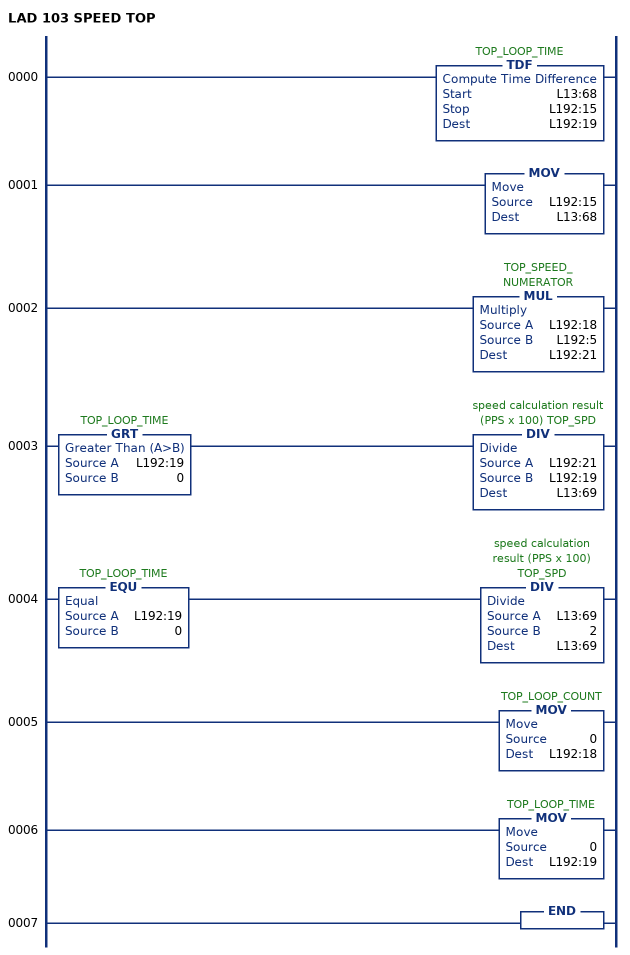
% Rung: 0 %
SOR TDF L13:68 L192:15 L192:19 EOR
%   L192:15  TOP_THIS_TIME  "rtc top belt movement event time" %
%   L192:19  TOP_LOOP_TIME %
% Rung: 1 %
SOR MOV L192:15 L13:68 EOR
%   L192:15  TOP_THIS_TIME  "rtc top belt movement event time" %
% Rung: 2 %
SOR MUL L192:18 L192:5 L192:21 EOR
%   L192:18  TOP_LOOP_COUNT %
%   L192:5  TKS_PER_SECOND %
%   L192:21  TOP_SPEED_NUMERATOR %
% Rung: 3 %
SOR GRT L192:19 0 DIV L192:21 L192:19 L13:69 EOR
%   L192:19  TOP_LOOP_TIME %
%   L192:21  TOP_SPEED_NUMERATOR %
%   L13:69  TOP_SPD  "speed calculation result (PPS x 100)" %
% Rung: 4 %
SOR EQU L192:19 0 DIV L13:69 2 L13:69 EOR
%   L192:19  TOP_LOOP_TIME %
%   L13:69  TOP_SPD  "speed calculation result (PPS x 100)" %
% Rung: 5 %
SOR MOV 0 L192:18 EOR
%   L192:18  TOP_LOOP_COUNT %
% Rung: 6 %
SOR MOV 0 L192:19 EOR
%   L192:19  TOP_LOOP_TIME %
% Rung: 7 %
SOR END EOR

LADDER 105 "P TOP"    % high speed %
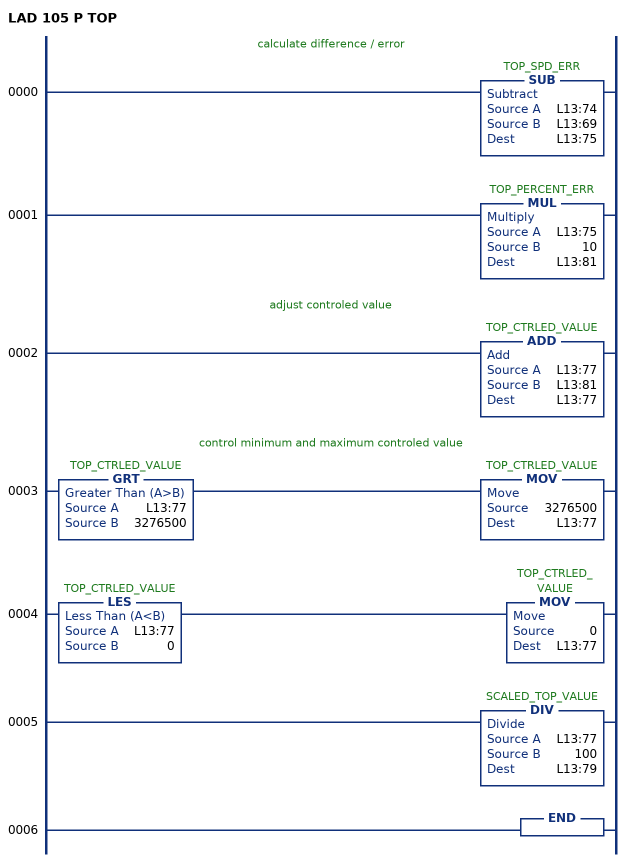
% Rung: 0 %
% calculate difference / error %
SOR SUB L13:74 L13:69 L13:75 EOR
%   L13:74  TOP_SPD_SETPOINT %
%   L13:69  TOP_SPD  "speed calculation result (PPS x 100)" %
%   L13:75  TOP_SPD_ERR %
% Rung: 1 %
SOR MUL L13:75 10 L13:81 EOR
%   L13:75  TOP_SPD_ERR %
%   L13:81  TOP_PERCENT_ERR %
% Rung: 2 %
% adjust controled value %
SOR ADD L13:77 L13:81 L13:77 EOR
%   L13:77  TOP_CTRLED_VALUE %
%   L13:81  TOP_PERCENT_ERR %
% Rung: 3 %
% control minimum and maximum controled value %
SOR GRT L13:77 3276500 MOV 3276500 L13:77 EOR
%   L13:77  TOP_CTRLED_VALUE %
% Rung: 4 %
SOR LES L13:77 0 MOV 0 L13:77 EOR
%   L13:77  TOP_CTRLED_VALUE %
% Rung: 5 %
SOR DIV L13:77 100 L13:79 EOR
%   L13:77  TOP_CTRLED_VALUE %
%   L13:79  SCALED_TOP_VALUE %
% Rung: 6 %
SOR END EOR

LADDER 111 "SHIFT TOP"
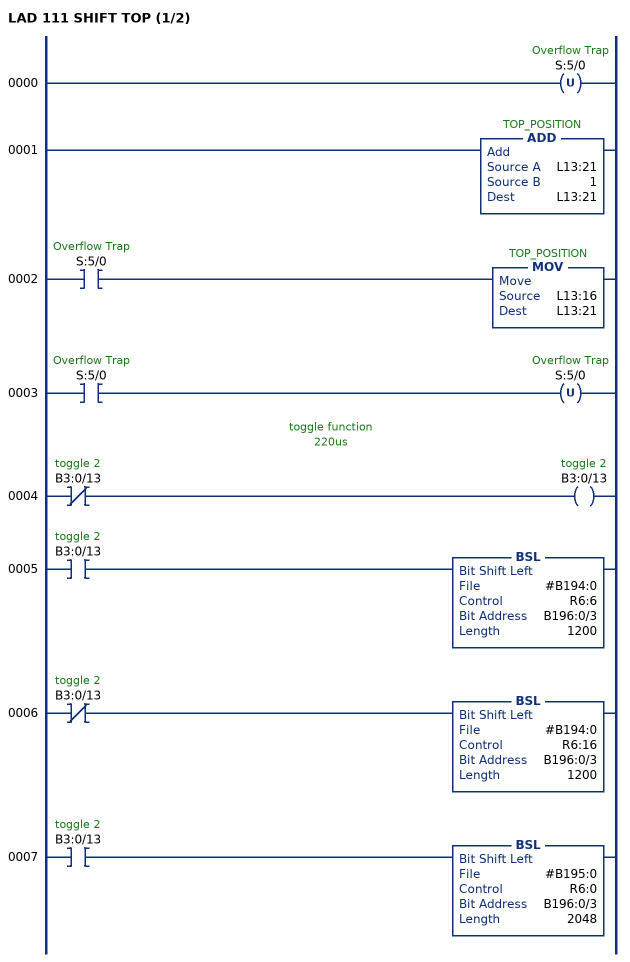
% Rung: 0 %
SOR OTU S:5/0 EOR
%   S:5/0  "Overflow Trap" %
% Rung: 1 %
SOR ADD L13:21 1 L13:21 EOR
%   L13:21  TOP_POSITION %
% Rung: 2 %
SOR XIC S:5/0 MOV L13:16 L13:21 EOR
%   S:5/0  "Overflow Trap" %
%   L13:16  MIN_LONG %
%   L13:21  TOP_POSITION %
% Rung: 3 %
SOR XIC S:5/0 OTU S:5/0 EOR
%   S:5/0  "Overflow Trap" %
% Rung: 4 %
% toggle function
% 220us %
SOR XIO B3:0/13 OTE B3:0/13 EOR
%   B3:0/13  "toggle 2" %
% Rung: 5 %
SOR XIC B3:0/13 BSL #B194:0 R6:6 B196:0/3 1200 EOR
%   B3:0/13  "toggle 2" %
%   R6:6  "from top load to top optic" %
%   B196:0/3  OFF %
% Rung: 6 %
SOR XIO B3:0/13 BSL #B194:0 R6:16 B196:0/3 1200 EOR
%   B3:0/13  "toggle 2" %
%   B196:0/3  OFF %
% Rung: 7 %
SOR XIC B3:0/13 BSL #B195:0 R6:0 B196:0/3 2048 EOR
%   B3:0/13  "toggle 2" %
%   B196:0/3  OFF %

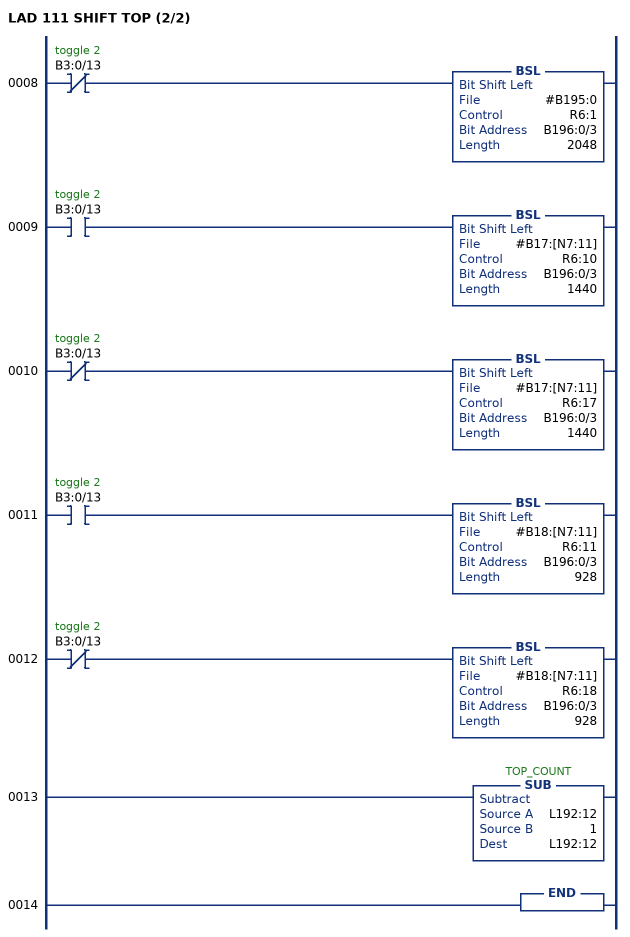
% Rung: 8 %
SOR XIO B3:0/13 BSL #B195:0 R6:1 B196:0/3 2048 EOR
%   B3:0/13  "toggle 2" %
%   B196:0/3  OFF %
% Rung: 9 %
SOR XIC B3:0/13 BSL #B17:[N7:11] R6:10 B196:0/3 1440 EOR
%   B3:0/13  "toggle 2" %
%   B196:0/3  OFF %
% Rung: 10 %
SOR XIO B3:0/13 BSL #B17:[N7:11] R6:17 B196:0/3 1440 EOR
%   B3:0/13  "toggle 2" %
%   B196:0/3  OFF %
% Rung: 11 %
SOR XIC B3:0/13 BSL #B18:[N7:11] R6:11 B196:0/3 928 EOR
%   B3:0/13  "toggle 2" %
%   B196:0/3  OFF %
% Rung: 12 %
SOR XIO B3:0/13 BSL #B18:[N7:11] R6:18 B196:0/3 928 EOR
%   B3:0/13  "toggle 2" %
%   B196:0/3  OFF %
% Rung: 13 %
SOR SUB L192:12 1 L192:12 EOR
%   L192:12  TOP_COUNT %
% Rung: 14 %
SOR END EOR

LADDER 131 "READXFER"
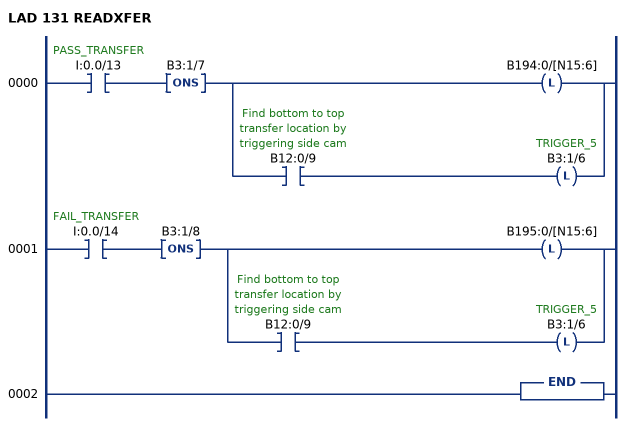
% Rung: 0 %
SOR XIC I:0.0/13 ONS B3:1/7 BST OTL B194:0/[N15:6] NXB XIC B12:0/9 OTL B3:1/6 BND EOR
%   I:0.0/13  PASS_TRANSFER %
%   N15:6  XFER_IN_LOC %
%   B12:0/9  "Find bottom to top transfer location by triggering side cam" %
%   B3:1/6  TRIGGER_5 %
% Rung: 1 %
SOR XIC I:0.0/14 ONS B3:1/8 BST OTL B195:0/[N15:6] NXB XIC B12:0/9 OTL B3:1/6 BND EOR
%   I:0.0/14  FAIL_TRANSFER %
%   N15:6  XFER_IN_LOC %
%   B12:0/9  "Find bottom to top transfer location by triggering side cam" %
%   B3:1/6  TRIGGER_5 %
% Rung: 2 %
SOR END EOR

LADDER 140 "TOP_OPTIC"
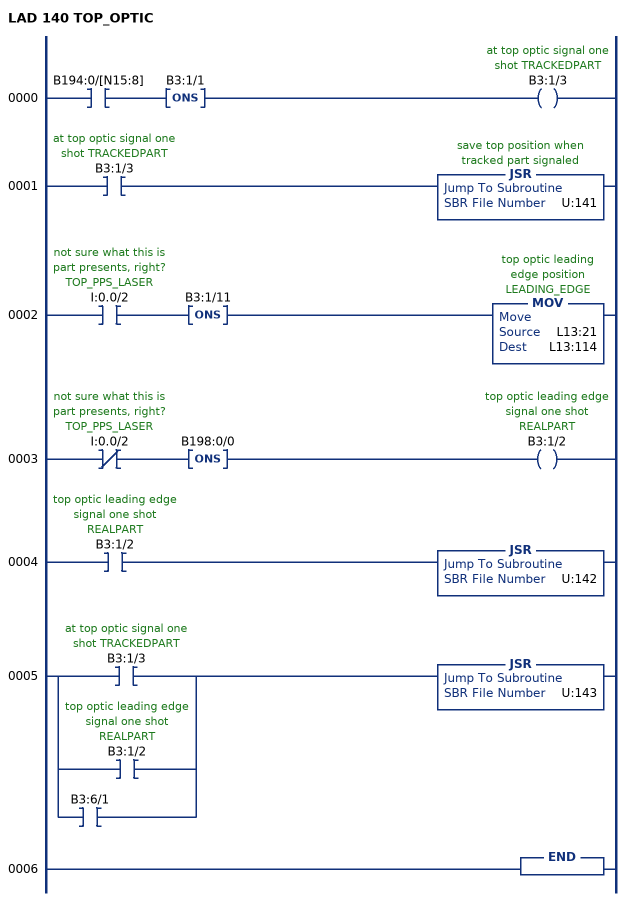
% Rung: 0 %
SOR XIC B194:0/[N15:8] ONS B3:1/1 OTE B3:1/3 EOR
%   N15:8  TOP_OPTIC_LOC %
%   B3:1/3  TRACKEDPART  "at top optic signal one shot" %
% Rung: 1 %
SOR XIC B3:1/3 JSR U:141 EOR
%   B3:1/3  TRACKEDPART  "at top optic signal one shot" %
%   U:141  "save top position when tracked part signaled" %
% Rung: 2 %
SOR XIC I:0.0/2 ONS B3:1/11 MOV L13:21 L13:114 EOR
%   I:0.0/2  TOP_PPS_LASER  "not sure what this is part presents, right?" %
%   L13:21  TOP_POSITION %
%   L13:114  LEADING_EDGE  "top optic leading edge position" %
% Rung: 3 %
SOR XIO I:0.0/2 ONS B198:0/0 OTE B3:1/2 EOR
%   I:0.0/2  TOP_PPS_LASER  "not sure what this is part presents, right?" %
%   B3:1/2  REALPART  "top optic leading edge signal one shot" %
% Rung: 4 %
SOR XIC B3:1/2 JSR U:142 EOR
%   B3:1/2  REALPART  "top optic leading edge signal one shot" %
% Rung: 5 %
SOR BST XIC B3:1/3 NXB XIC B3:1/2 NXB XIC B3:6/1 BND JSR U:143 EOR
%   B3:1/3  TRACKEDPART  "at top optic signal one shot" %
%   B3:1/2  REALPART  "top optic leading edge signal one shot" %
% Rung: 6 %
SOR END EOR

LADDER 141 "TOPOP_VERT"
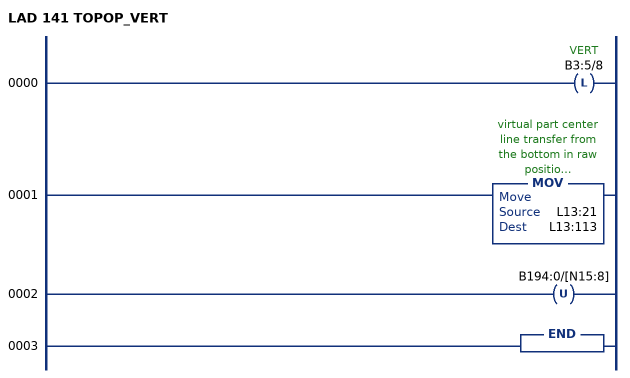
% Rung: 0 %
SOR OTL B3:5/8 EOR
%   B3:5/8  VERT %
% Rung: 1 %
SOR MOV L13:21 L13:113 EOR
%   L13:21  TOP_POSITION %
%   L13:113  VERTUAL_PT_RAW_CL  "virtual part center line transfer from the bottom in raw position" %
% Rung: 2 %
SOR OTU B194:0/[N15:8] EOR
%   N15:8  TOP_OPTIC_LOC %
% Rung: 3 %
SOR END EOR

LADDER 142 "TOPOP_REAL"
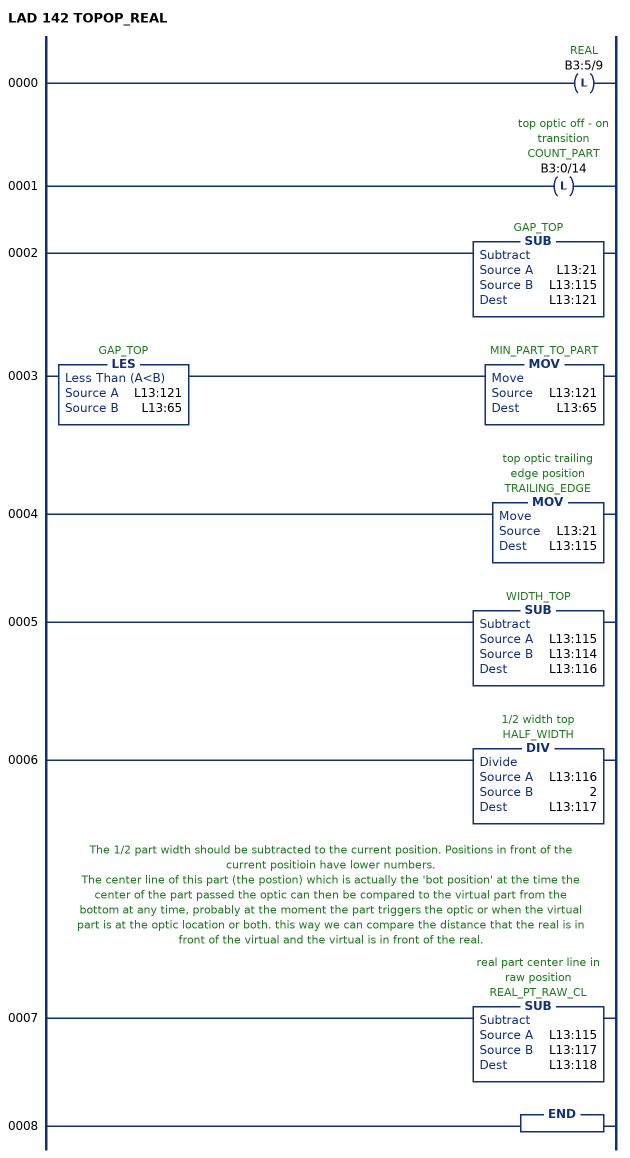
% Rung: 0 %
SOR OTL B3:5/9 EOR
%   B3:5/9  REAL %
% Rung: 1 %
SOR OTL B3:0/14 EOR
%   B3:0/14  COUNT_PART  "top optic off - on transition" %
% Rung: 2 %
SOR SUB L13:21 L13:115 L13:121 EOR
%   L13:21  TOP_POSITION %
%   L13:115  TRAILING_EDGE  "top optic trailing edge position" %
%   L13:121  GAP_TOP %
% Rung: 3 %
SOR LES L13:121 L13:65 MOV L13:121 L13:65 EOR
%   L13:121  GAP_TOP %
%   L13:65  MIN_PART_TO_PART %
% Rung: 4 %
SOR MOV L13:21 L13:115 EOR
%   L13:21  TOP_POSITION %
%   L13:115  TRAILING_EDGE  "top optic trailing edge position" %
% Rung: 5 %
SOR SUB L13:115 L13:114 L13:116 EOR
%   L13:115  TRAILING_EDGE  "top optic trailing edge position" %
%   L13:114  LEADING_EDGE  "top optic leading edge position" %
%   L13:116  WIDTH_TOP %
% Rung: 6 %
SOR DIV L13:116 2 L13:117 EOR
%   L13:116  WIDTH_TOP %
%   L13:117  HALF_WIDTH  "1/2 width top" %
% Rung: 7 %
% The 1/2 part width should be subtracted to the current position. Positions in front of the current positioin have lower numbers.
% 
% The center line of this part (the postion) which is actually the 'bot position' at the time the center of the part passed the optic can then be compared to the virtual part from the bottom at any time, probably at the moment the part triggers the optic or when the virtual part is at the optic location or both. this way we can compare the distance that the real is in front of the virtual and the virtual is in front of the real. %
SOR SUB L13:115 L13:117 L13:118 EOR
%   L13:115  TRAILING_EDGE  "top optic trailing edge position" %
%   L13:117  HALF_WIDTH  "1/2 width top" %
%   L13:118  REAL_PT_RAW_CL  "real part center line in raw position" %
% Rung: 8 %
SOR END EOR

LADDER 143 "TOPOP_TEST"
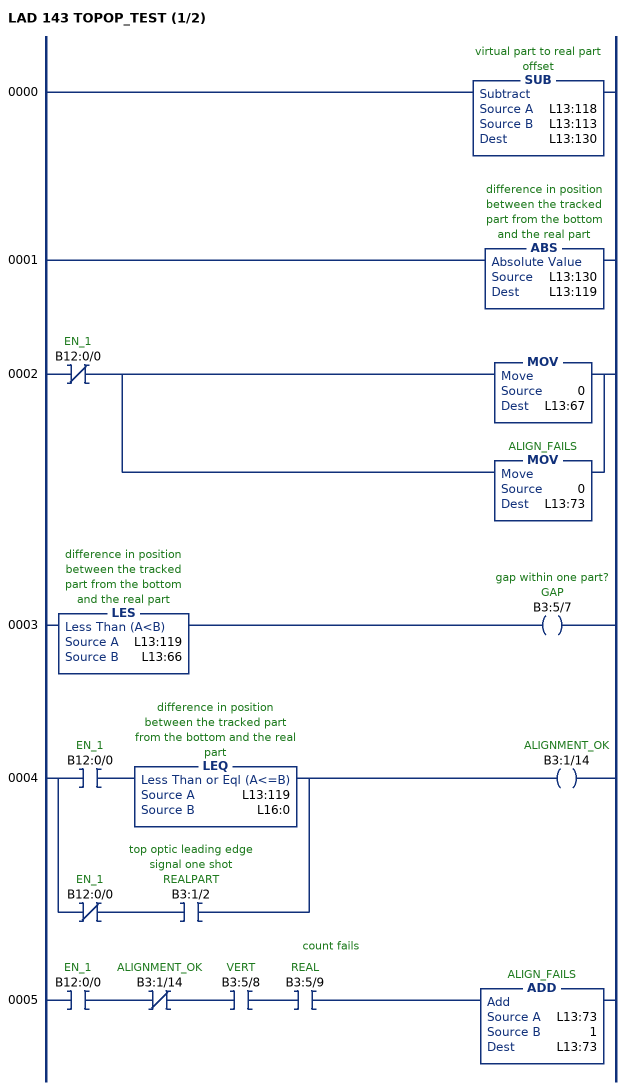
% Rung: 0 %
SOR SUB L13:118 L13:113 L13:130 EOR
%   L13:118  REAL_PT_RAW_CL  "real part center line in raw position" %
%   L13:113  VERTUAL_PT_RAW_CL  "virtual part center line transfer from the bottom in raw position" %
%   L13:130  "virtual part to real part offset" %
% Rung: 1 %
SOR ABS L13:130 L13:119 EOR
%   L13:130  "virtual part to real part offset" %
%   L13:119  "difference in position between the tracked part from the bottom and the real part" %
% Rung: 2 %
SOR XIO B12:0/0 BST MOV 0 L13:67 NXB MOV 0 L13:73 BND EOR
%   B12:0/0  EN_1 %
%   L13:73  ALIGN_FAILS %
% Rung: 3 %
SOR LES L13:119 L13:66 OTE B3:5/7 EOR
%   L13:119  "difference in position between the tracked part from the bottom and the real part" %
%   L13:66  SAME_PART_GAP %
%   B3:5/7  GAP  "gap within one part?" %
% Rung: 4 %
SOR BST XIC B12:0/0 LEQ L13:119 L16:0 NXB XIO B12:0/0 XIC B3:1/2 BND OTE B3:1/14 EOR
%   B12:0/0  EN_1 %
%   L13:119  "difference in position between the tracked part from the bottom and the real part" %
%   L16:0  MAX_OFFSET %
%   B3:1/2  REALPART  "top optic leading edge signal one shot" %
%   B3:1/14  ALIGNMENT_OK %
% Rung: 5 %
% count fails %
SOR XIC B12:0/0 XIO B3:1/14 XIC B3:5/8 XIC B3:5/9 ADD L13:73 1 L13:73 EOR
%   B12:0/0  EN_1 %
%   B3:1/14  ALIGNMENT_OK %
%   B3:5/8  VERT %
%   B3:5/9  REAL %
%   L13:73  ALIGN_FAILS %

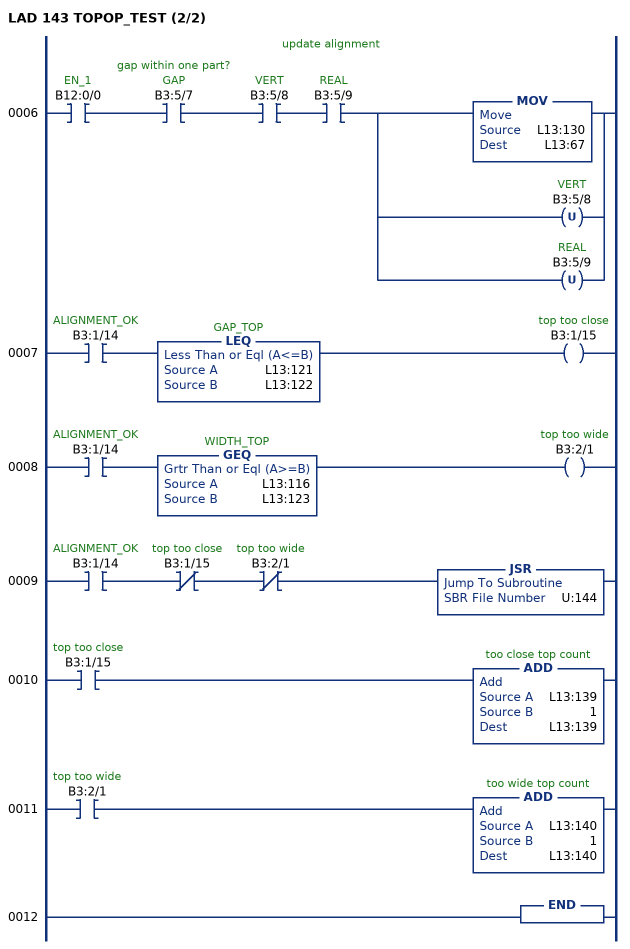
% Rung: 6 %
% update alignment %
SOR XIC B12:0/0 XIC B3:5/7 XIC B3:5/8 XIC B3:5/9 BST MOV L13:130 L13:67 NXB OTU B3:5/8 NXB OTU B3:5/9 BND EOR
%   B12:0/0  EN_1 %
%   B3:5/7  GAP  "gap within one part?" %
%   B3:5/8  VERT %
%   B3:5/9  REAL %
%   L13:130  "virtual part to real part offset" %
% Rung: 7 %
SOR XIC B3:1/14 LEQ L13:121 L13:122 OTE B3:1/15 EOR
%   B3:1/14  ALIGNMENT_OK %
%   L13:121  GAP_TOP %
%   L13:122  MIN_GAP_TOP %
%   B3:1/15  "top too close" %
% Rung: 8 %
SOR XIC B3:1/14 GEQ L13:116 L13:123 OTE B3:2/1 EOR
%   B3:1/14  ALIGNMENT_OK %
%   L13:116  WIDTH_TOP %
%   L13:123  MAX_WIDTH_TOP %
%   B3:2/1  "top too wide" %
% Rung: 9 %
SOR XIC B3:1/14 XIO B3:1/15 XIO B3:2/1 JSR U:144 EOR
%   B3:1/14  ALIGNMENT_OK %
%   B3:1/15  "top too close" %
%   B3:2/1  "top too wide" %
% Rung: 10 %
SOR XIC B3:1/15 ADD L13:139 1 L13:139 EOR
%   B3:1/15  "top too close" %
%   L13:139  "too close top count" %
% Rung: 11 %
SOR XIC B3:2/1 ADD L13:140 1 L13:140 EOR
%   B3:2/1  "top too wide" %
%   L13:140  "too wide top count" %
% Rung: 12 %
SOR END EOR

LADDER 144 "TOP_OP_OK"
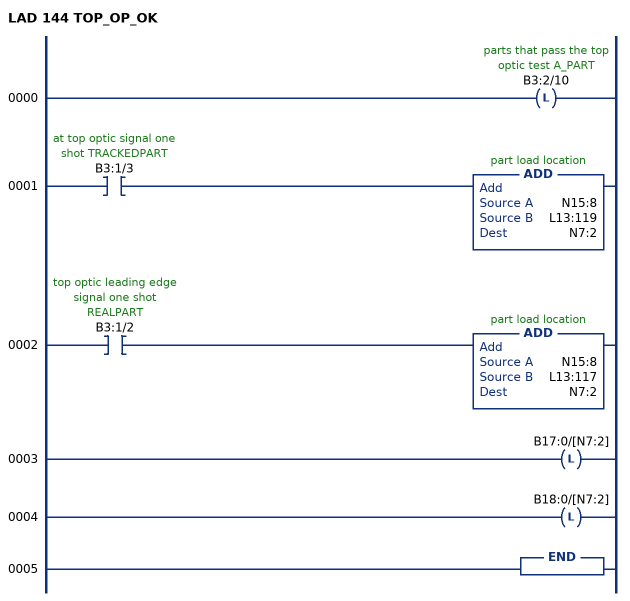
% Rung: 0 %
SOR OTL B3:2/10 EOR
%   B3:2/10  A_PART  "parts that pass the top optic test" %
% Rung: 1 %
SOR XIC B3:1/3 ADD N15:8 L13:119 N7:2 EOR
%   B3:1/3  TRACKEDPART  "at top optic signal one shot" %
%   N15:8  TOP_OPTIC_LOC %
%   L13:119  "difference in position between the tracked part from the bottom and the real part" %
%   N7:2  "part load location" %
% Rung: 2 %
SOR XIC B3:1/2 ADD N15:8 L13:117 N7:2 EOR
%   B3:1/2  REALPART  "top optic leading edge signal one shot" %
%   N15:8  TOP_OPTIC_LOC %
%   L13:117  HALF_WIDTH  "1/2 width top" %
%   N7:2  "part load location" %
% Rung: 3 %
SOR OTL B17:0/[N7:2] EOR
%   N7:2  "part load location" %
% Rung: 4 %
SOR OTL B18:0/[N7:2] EOR
%   N7:2  "part load location" %
% Rung: 5 %
SOR END EOR

LADDER 190 "INS5"
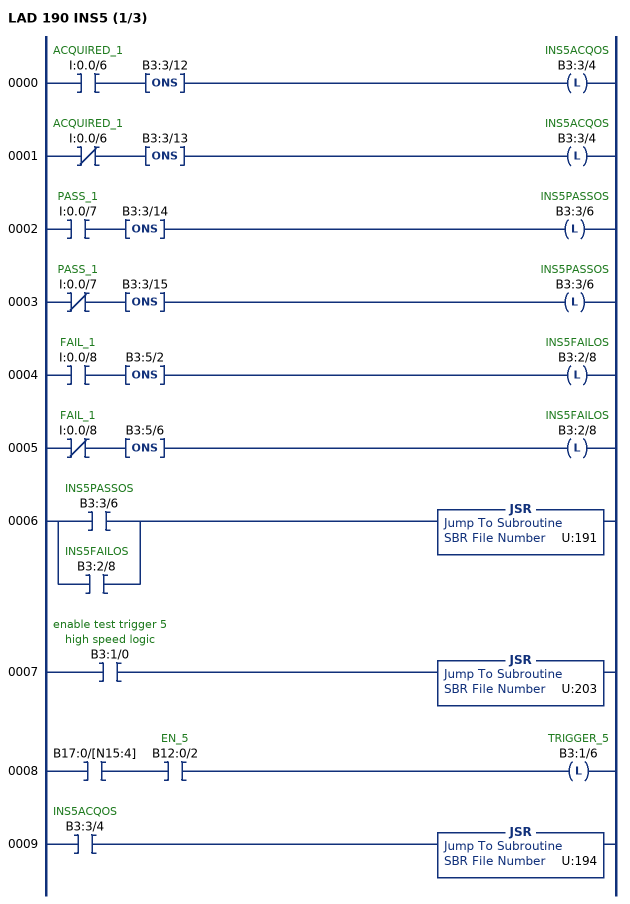
% Rung: 0 %
SOR XIC I:0.0/6 ONS B3:3/12 OTL B3:3/4 EOR
%   I:0.0/6  ACQUIRED_1 %
%   B3:3/4  INS5ACQOS %
% Rung: 1 %
SOR XIO I:0.0/6 ONS B3:3/13 OTL B3:3/4 EOR
%   I:0.0/6  ACQUIRED_1 %
%   B3:3/4  INS5ACQOS %
% Rung: 2 %
SOR XIC I:0.0/7 ONS B3:3/14 OTL B3:3/6 EOR
%   I:0.0/7  PASS_1 %
%   B3:3/6  INS5PASSOS %
% Rung: 3 %
SOR XIO I:0.0/7 ONS B3:3/15 OTL B3:3/6 EOR
%   I:0.0/7  PASS_1 %
%   B3:3/6  INS5PASSOS %
% Rung: 4 %
SOR XIC I:0.0/8 ONS B3:5/2 OTL B3:2/8 EOR
%   I:0.0/8  FAIL_1 %
%   B3:2/8  INS5FAILOS %
% Rung: 5 %
SOR XIO I:0.0/8 ONS B3:5/6 OTL B3:2/8 EOR
%   I:0.0/8  FAIL_1 %
%   B3:2/8  INS5FAILOS %
% Rung: 6 %
SOR BST XIC B3:3/6 NXB XIC B3:2/8 BND JSR U:191 EOR
%   B3:3/6  INS5PASSOS %
%   B3:2/8  INS5FAILOS %
% Rung: 7 %
SOR XIC B3:1/0 JSR U:203 EOR
%   B3:1/0  "enable test trigger 5 high speed logic" %
% Rung: 8 %
SOR XIC B17:0/[N15:4] XIC B12:0/2 OTL B3:1/6 EOR
%   N15:4  INS_5_TRIG_LOC %
%   B12:0/2  EN_5 %
%   B3:1/6  TRIGGER_5 %
% Rung: 9 %
SOR XIC B3:3/4 JSR U:194 EOR
%   B3:3/4  INS5ACQOS %

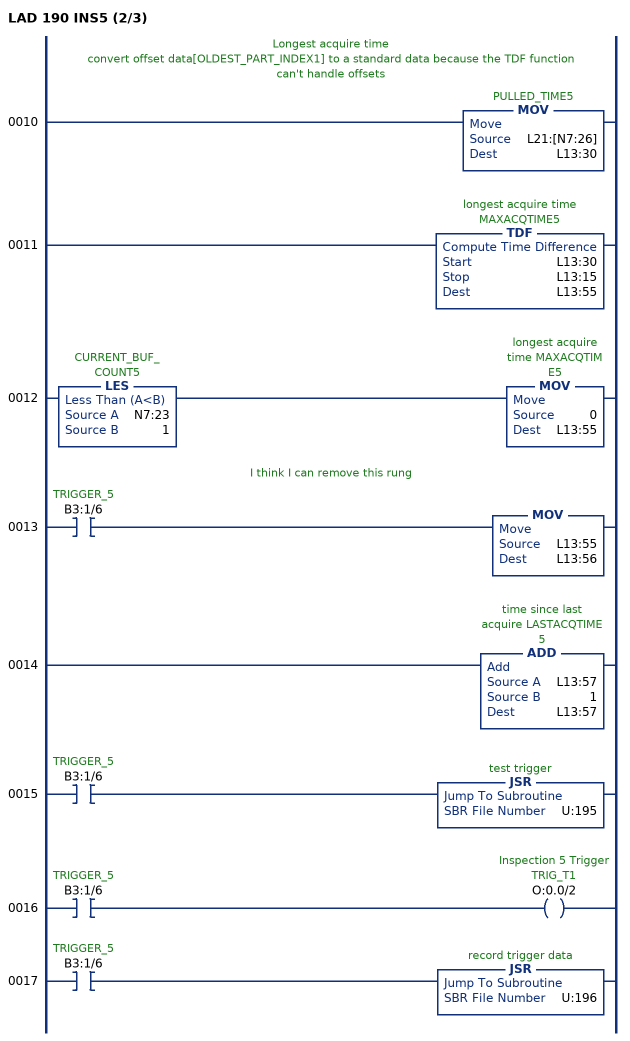
% Rung: 10 %
% Longest acquire time
% convert offset data[OLDEST_PART_INDEX1] to a standard data because the TDF function can't handle offsets %
SOR MOV L21:[N7:26] L13:30 EOR
%   N7:26  OLDEST_PART_INDEX5 %
%   L13:30  PULLED_TIME5 %
% Rung: 11 %
SOR TDF L13:30 L13:15 L13:55 EOR
%   L13:30  PULLED_TIME5 %
%   L13:15  TOP_TIME %
%   L13:55  MAXACQTIME5  "longest acquire time" %
% Rung: 12 %
SOR LES N7:23 1 MOV 0 L13:55 EOR
%   N7:23  CURRENT_BUF_COUNT5 %
%   L13:55  MAXACQTIME5  "longest acquire time" %
% Rung: 13 %
% I think I can remove this rung %
SOR XIC B3:1/6 MOV L13:55 L13:56 EOR
%   B3:1/6  TRIGGER_5 %
%   L13:55  MAXACQTIME5  "longest acquire time" %
% Rung: 14 %
SOR ADD L13:57 1 L13:57 EOR
%   L13:57  LASTACQTIME5  "time since last acquire" %
% Rung: 15 %
SOR XIC B3:1/6 JSR U:195 EOR
%   B3:1/6  TRIGGER_5 %
%   U:195  "test trigger" %
% Rung: 16 %
SOR XIC B3:1/6 OTE O:0.0/2 EOR
%   B3:1/6  TRIGGER_5 %
%   O:0.0/2  TRIG_T1  "Inspection 5 Trigger" %
% Rung: 17 %
SOR XIC B3:1/6 JSR U:196 EOR
%   B3:1/6  TRIGGER_5 %
%   U:196  "record trigger data" %

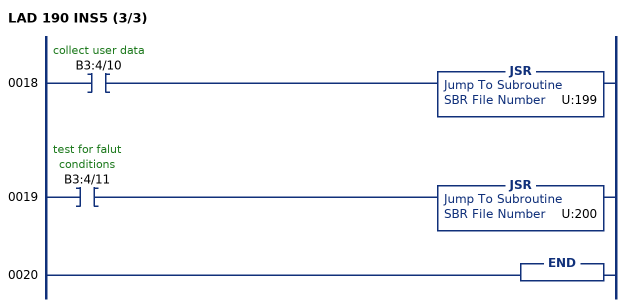
% Rung: 18 %
SOR XIC B3:4/10 JSR U:199 EOR
%   B3:4/10  "collect user data" %
% Rung: 19 %
SOR XIC B3:4/11 JSR U:200 EOR
%   B3:4/11  "test for falut conditions" %
% Rung: 20 %
SOR END EOR

LADDER 191 "INS5RESULT"
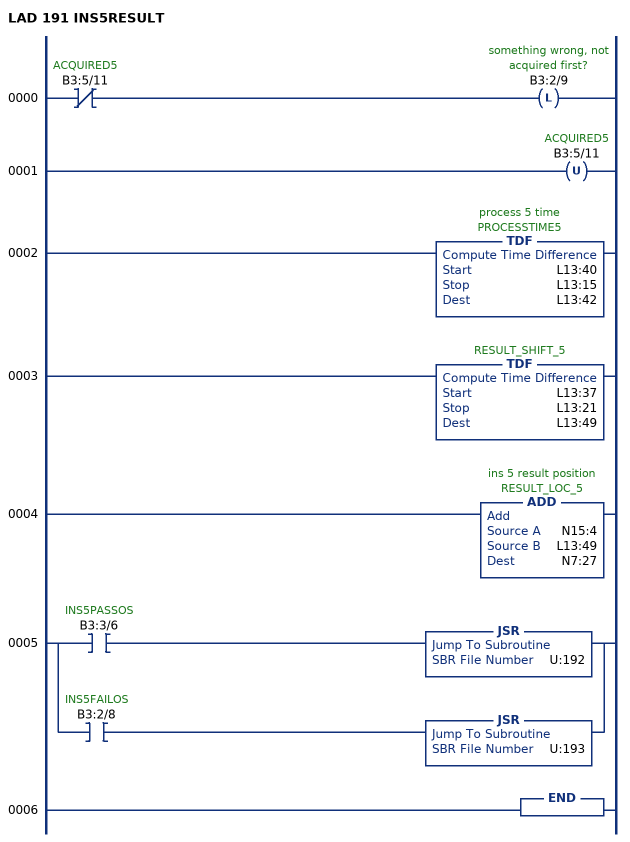
% Rung: 0 %
SOR XIO B3:5/11 OTL B3:2/9 EOR
%   B3:5/11  ACQUIRED5 %
%   B3:2/9  "something wrong, not acquired first?" %
% Rung: 1 %
SOR OTU B3:5/11 EOR
%   B3:5/11  ACQUIRED5 %
% Rung: 2 %
SOR TDF L13:40 L13:15 L13:42 EOR
%   L13:40  TIMEOFACQ5  "the time of the last acquire" %
%   L13:15  TOP_TIME %
%   L13:42  PROCESSTIME5  "process 5 time" %
% Rung: 3 %
SOR TDF L13:37 L13:21 L13:49 EOR
%   L13:37  PROCESS_START_POS_5 %
%   L13:21  TOP_POSITION %
%   L13:49  RESULT_SHIFT_5 %
% Rung: 4 %
SOR ADD N15:4 L13:49 N7:27 EOR
%   N15:4  INS_5_TRIG_LOC %
%   L13:49  RESULT_SHIFT_5 %
%   N7:27  RESULT_LOC_5  "ins 5 result position" %
% Rung: 5 %
SOR BST XIC B3:3/6 JSR U:192 NXB XIC B3:2/8 JSR U:193 BND EOR
%   B3:3/6  INS5PASSOS %
%   B3:2/8  INS5FAILOS %
% Rung: 6 %
SOR END EOR

LADDER 192 "INS5PASS"
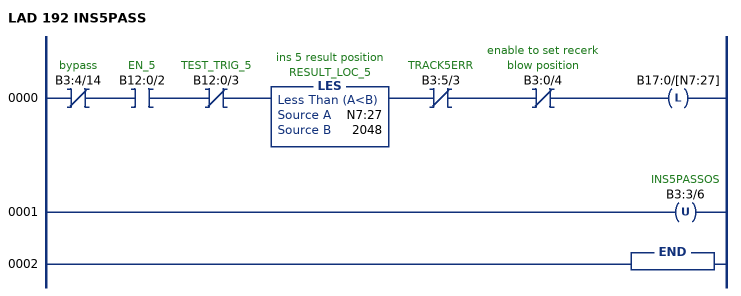
% Rung: 0 %
SOR XIO B3:4/14 XIC B12:0/2 XIO B12:0/3 LES N7:27 2048 XIO B3:5/3 XIO B3:0/4 OTL B17:0/[N7:27] EOR
%   B3:4/14  "bypass" %
%   B12:0/2  EN_5 %
%   B12:0/3  TEST_TRIG_5 %
%   N7:27  RESULT_LOC_5  "ins 5 result position" %
%   B3:5/3  TRACK5ERR %
%   B3:0/4  "enable to set recerk blow position" %
% Rung: 1 %
SOR OTU B3:3/6 EOR
%   B3:3/6  INS5PASSOS %
% Rung: 2 %
SOR END EOR

LADDER 193 "INS5FAIL"
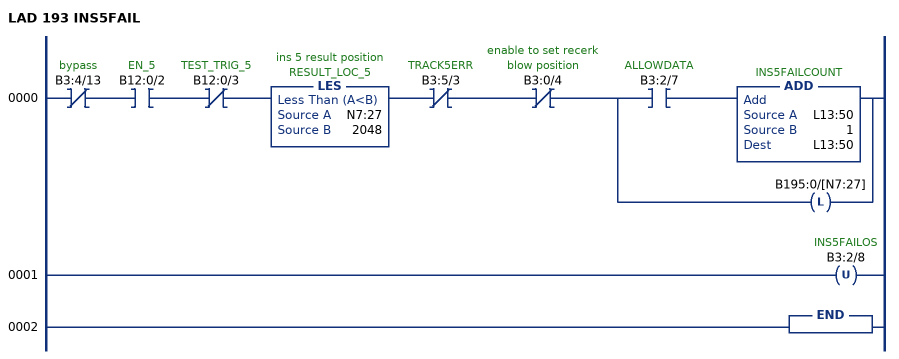
% Rung: 0 %
SOR XIO B3:4/13 XIC B12:0/2 XIO B12:0/3 LES N7:27 2048 XIO B3:5/3 XIO B3:0/4 BST XIC B3:2/7 ADD L13:50 1 L13:50 NXB OTL B195:0/[N7:27] BND EOR
%   B3:4/13  "bypass" %
%   B12:0/2  EN_5 %
%   B12:0/3  TEST_TRIG_5 %
%   N7:27  RESULT_LOC_5  "ins 5 result position" %
%   B3:5/3  TRACK5ERR %
%   B3:0/4  "enable to set recerk blow position" %
%   B3:2/7  ALLOWDATA %
%   L13:50  INS5FAILCOUNT %
% Rung: 1 %
SOR OTU B3:2/8 EOR
%   B3:2/8  INS5FAILOS %
% Rung: 2 %
SOR END EOR

LADDER 194 "INS5ACQ"
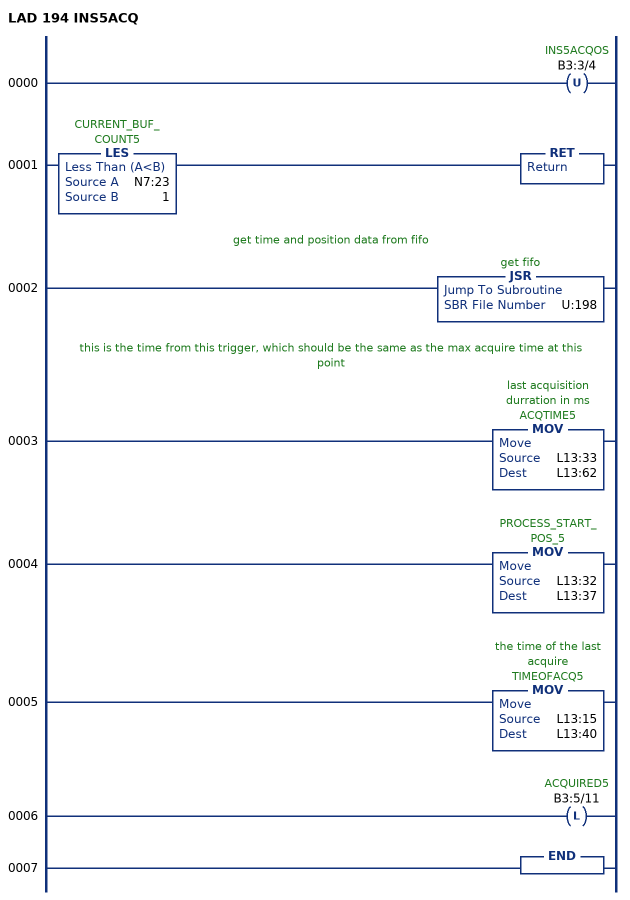
% Rung: 0 %
SOR OTU B3:3/4 EOR
%   B3:3/4  INS5ACQOS %
% Rung: 1 %
SOR LES N7:23 1 RET EOR
%   N7:23  CURRENT_BUF_COUNT5 %
% Rung: 2 %
% get time and position data from fifo %
SOR JSR U:198 EOR
%   U:198  "get fifo" %
% Rung: 3 %
% this is the time from this trigger, which should be the same as the max acquire time at this point %
SOR MOV L13:33 L13:62 EOR
%   L13:33  TIME_SPAN5 %
%   L13:62  ACQTIME5  "last acquisition durration in ms" %
% Rung: 4 %
SOR MOV L13:32 L13:37 EOR
%   L13:32  PULLED_POSITION5 %
%   L13:37  PROCESS_START_POS_5 %
% Rung: 5 %
SOR MOV L13:15 L13:40 EOR
%   L13:15  TOP_TIME %
%   L13:40  TIMEOFACQ5  "the time of the last acquire" %
% Rung: 6 %
SOR OTL B3:5/11 EOR
%   B3:5/11  ACQUIRED5 %
% Rung: 7 %
SOR END EOR

LADDER 195 "Q5TIMETEST"
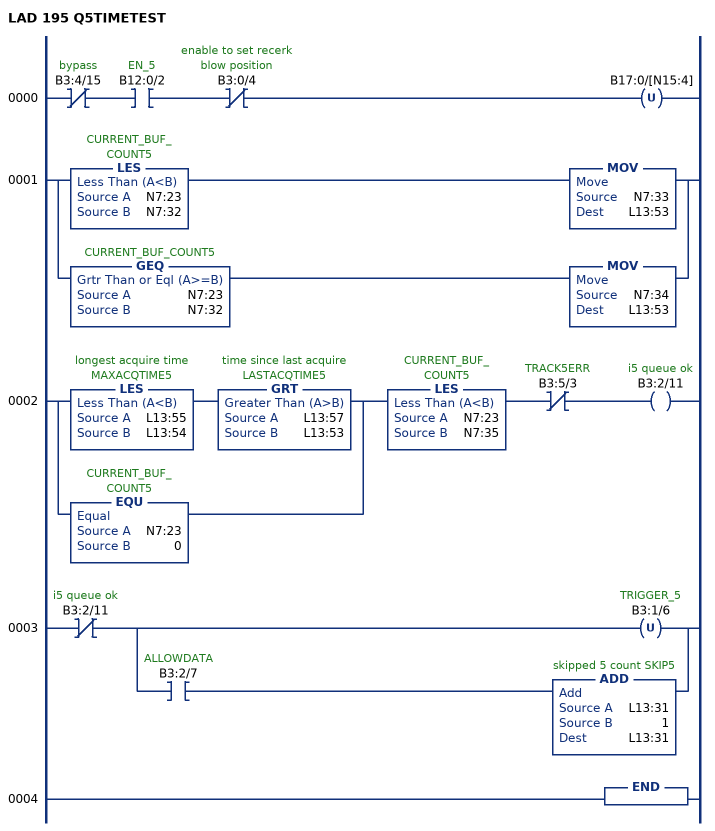
% Rung: 0 %
SOR XIO B3:4/15 XIC B12:0/2 XIO B3:0/4 OTU B17:0/[N15:4] EOR
%   B3:4/15  "bypass" %
%   B12:0/2  EN_5 %
%   B3:0/4  "enable to set recerk blow position" %
%   N15:4  INS_5_TRIG_LOC %
% Rung: 1 %
SOR BST LES N7:23 N7:32 MOV N7:33 L13:53 NXB GEQ N7:23 N7:32 MOV N7:34 L13:53 BND EOR
%   N7:23  CURRENT_BUF_COUNT5 %
% Rung: 2 %
SOR BST LES L13:55 L13:54 GRT L13:57 L13:53 NXB EQU N7:23 0 BND LES N7:23 N7:35 XIO B3:5/3 OTE B3:2/11 EOR
%   L13:55  MAXACQTIME5  "longest acquire time" %
%   L13:57  LASTACQTIME5  "time since last acquire" %
%   N7:23  CURRENT_BUF_COUNT5 %
%   N7:35  "maximum buffers" %
%   B3:5/3  TRACK5ERR %
%   B3:2/11  "i5 queue ok" %
% Rung: 3 %
SOR XIO B3:2/11 BST OTU B3:1/6 NXB XIC B3:2/7 ADD L13:31 1 L13:31 BND EOR
%   B3:2/11  "i5 queue ok" %
%   B3:1/6  TRIGGER_5 %
%   B3:2/7  ALLOWDATA %
%   L13:31  SKIP5  "skipped 5 count" %
% Rung: 4 %
SOR END EOR

LADDER 196 "INS5TRIG"
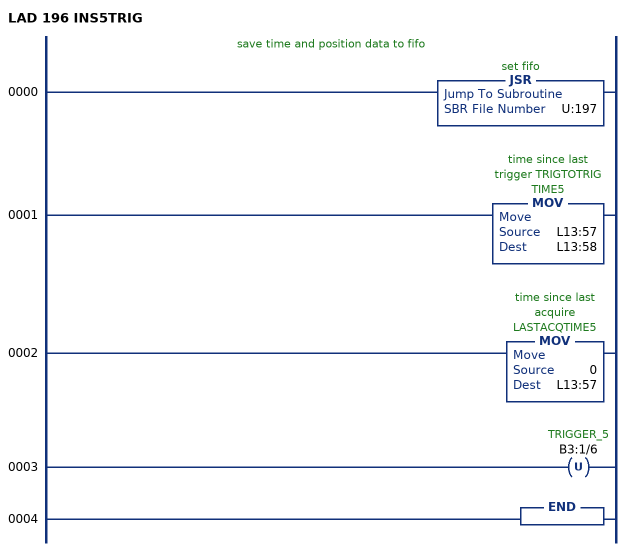
% Rung: 0 %
% save time and position data to fifo %
SOR JSR U:197 EOR
%   U:197  "set fifo" %
% Rung: 1 %
SOR MOV L13:57 L13:58 EOR
%   L13:57  LASTACQTIME5  "time since last acquire" %
%   L13:58  TRIGTOTRIGTIME5  "time since last trigger" %
% Rung: 2 %
SOR MOV 0 L13:57 EOR
%   L13:57  LASTACQTIME5  "time since last acquire" %
% Rung: 3 %
SOR OTU B3:1/6 EOR
%   B3:1/6  TRIGGER_5 %
% Rung: 4 %
SOR END EOR

LADDER 197 "FIFO5SET"
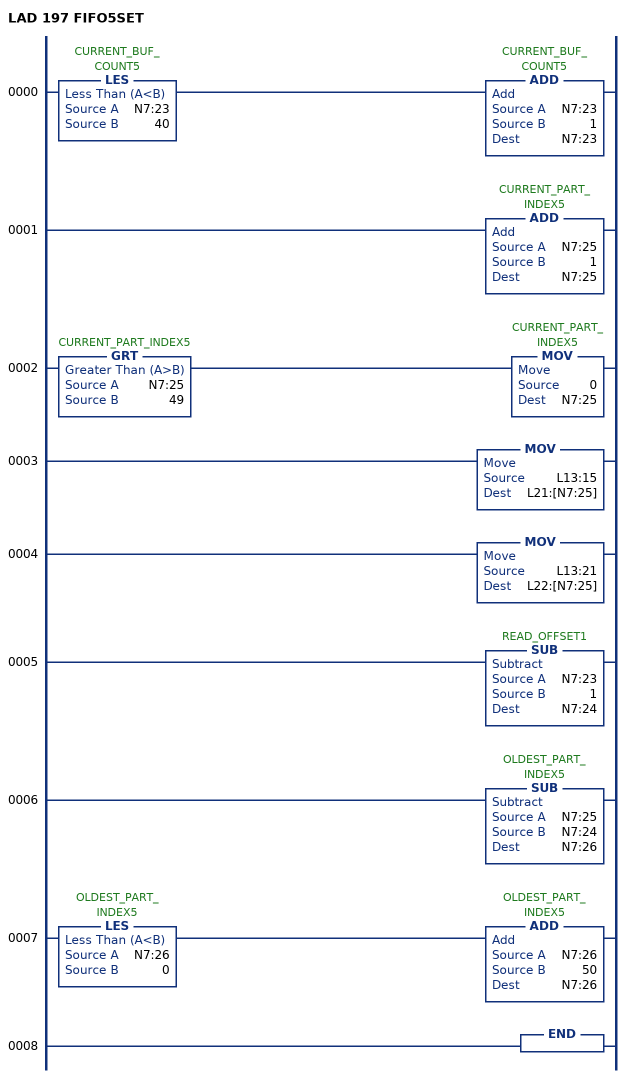
% Rung: 0 %
SOR LES N7:23 40 ADD N7:23 1 N7:23 EOR
%   N7:23  CURRENT_BUF_COUNT5 %
% Rung: 1 %
SOR ADD N7:25 1 N7:25 EOR
%   N7:25  CURRENT_PART_INDEX5 %
% Rung: 2 %
SOR GRT N7:25 49 MOV 0 N7:25 EOR
%   N7:25  CURRENT_PART_INDEX5 %
% Rung: 3 %
SOR MOV L13:15 L21:[N7:25] EOR
%   L13:15  TOP_TIME %
%   N7:25  CURRENT_PART_INDEX5 %
% Rung: 4 %
SOR MOV L13:21 L22:[N7:25] EOR
%   L13:21  TOP_POSITION %
%   N7:25  CURRENT_PART_INDEX5 %
% Rung: 5 %
SOR SUB N7:23 1 N7:24 EOR
%   N7:23  CURRENT_BUF_COUNT5 %
%   N7:24  "READ_OFFSET1" %
% Rung: 6 %
SOR SUB N7:25 N7:24 N7:26 EOR
%   N7:25  CURRENT_PART_INDEX5 %
%   N7:24  "READ_OFFSET1" %
%   N7:26  OLDEST_PART_INDEX5 %
% Rung: 7 %
SOR LES N7:26 0 ADD N7:26 50 N7:26 EOR
%   N7:26  OLDEST_PART_INDEX5 %
% Rung: 8 %
SOR END EOR

LADDER 198 "FIFO5GET"
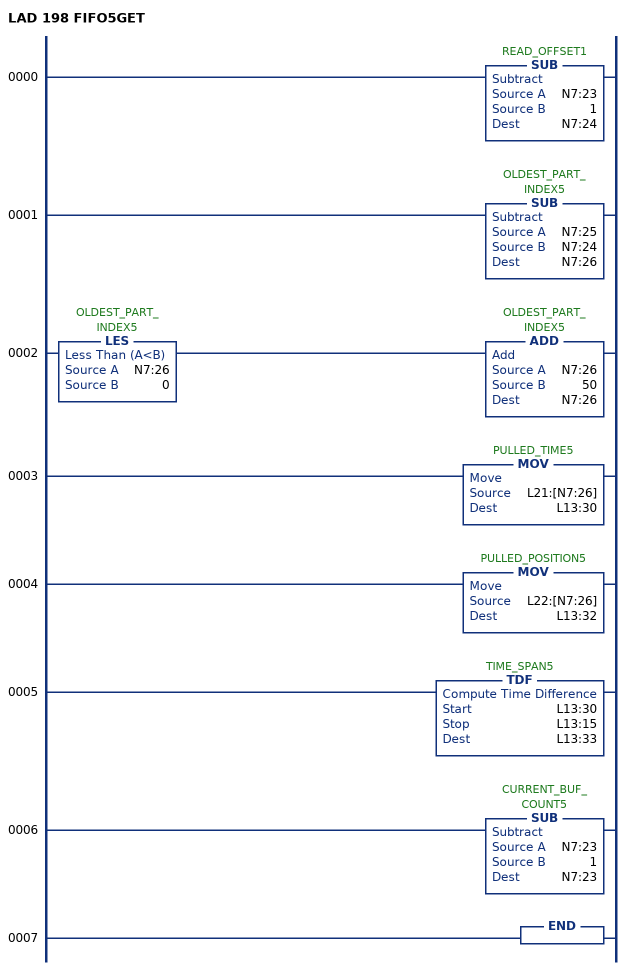
% Rung: 0 %
SOR SUB N7:23 1 N7:24 EOR
%   N7:23  CURRENT_BUF_COUNT5 %
%   N7:24  "READ_OFFSET1" %
% Rung: 1 %
SOR SUB N7:25 N7:24 N7:26 EOR
%   N7:25  CURRENT_PART_INDEX5 %
%   N7:24  "READ_OFFSET1" %
%   N7:26  OLDEST_PART_INDEX5 %
% Rung: 2 %
SOR LES N7:26 0 ADD N7:26 50 N7:26 EOR
%   N7:26  OLDEST_PART_INDEX5 %
% Rung: 3 %
SOR MOV L21:[N7:26] L13:30 EOR
%   N7:26  OLDEST_PART_INDEX5 %
%   L13:30  PULLED_TIME5 %
% Rung: 4 %
SOR MOV L22:[N7:26] L13:32 EOR
%   N7:26  OLDEST_PART_INDEX5 %
%   L13:32  PULLED_POSITION5 %
% Rung: 5 %
SOR TDF L13:30 L13:15 L13:33 EOR
%   L13:30  PULLED_TIME5 %
%   L13:15  TOP_TIME %
%   L13:33  TIME_SPAN5 %
% Rung: 6 %
SOR SUB N7:23 1 N7:23 EOR
%   N7:23  CURRENT_BUF_COUNT5 %
% Rung: 7 %
SOR END EOR

LADDER 199 "INSDATA5"
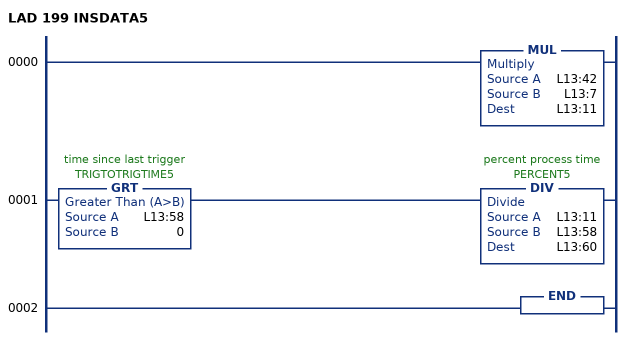
% Rung: 0 %
SOR MUL L13:42 L13:7 L13:11 EOR
%   L13:42  PROCESSTIME5  "process 5 time" %
% Rung: 1 %
SOR GRT L13:58 0 DIV L13:11 L13:58 L13:60 EOR
%   L13:58  TRIGTOTRIGTIME5  "time since last trigger" %
%   L13:60  PERCENT5  "percent process time" %
% Rung: 2 %
SOR END EOR

LADDER 200 "TESTFAULT5"
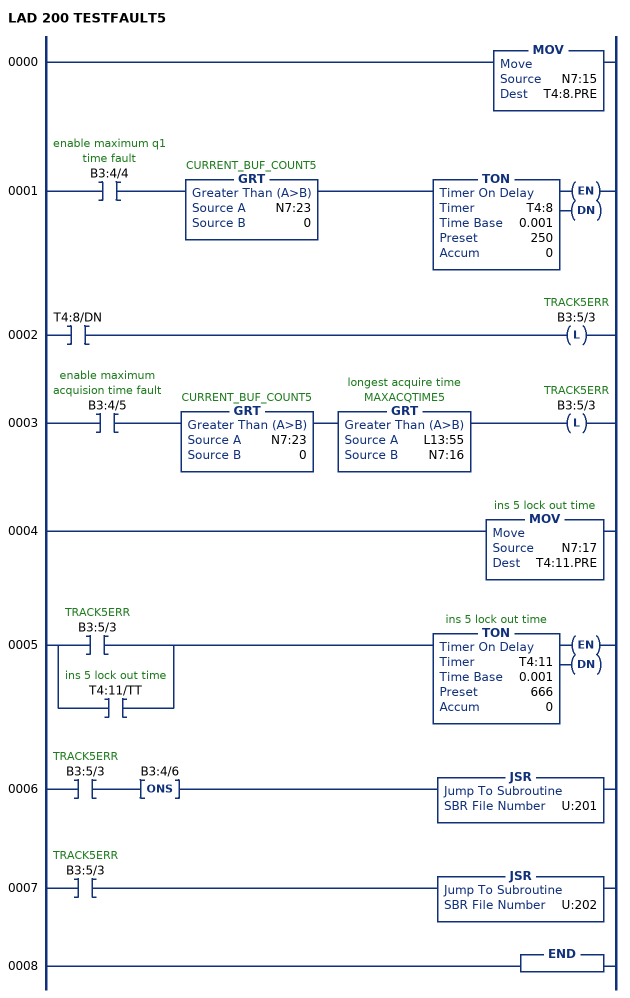
% Rung: 0 %
SOR MOV N7:15 T4:8.PRE EOR
%   N7:15  "max allowed ms time for q to be above 1 if safe fault is used" %
% Rung: 1 %
SOR XIC B3:4/4 GRT N7:23 0 TON T4:8 0.001 250 0 EOR
%   B3:4/4  "enable maximum q1 time fault" %
%   N7:23  CURRENT_BUF_COUNT5 %
% Rung: 2 %
SOR XIC T4:8/DN OTL B3:5/3 EOR
%   B3:5/3  TRACK5ERR %
% Rung: 3 %
SOR XIC B3:4/5 GRT N7:23 0 GRT L13:55 N7:16 OTL B3:5/3 EOR
%   B3:4/5  "enable maximum acquision time fault" %
%   N7:23  CURRENT_BUF_COUNT5 %
%   L13:55  MAXACQTIME5  "longest acquire time" %
%   N7:16  "maximum of the longest acquire time allowed if maximum acquire time fault is enabled" %
%   B3:5/3  TRACK5ERR %
% Rung: 4 %
SOR MOV N7:17 T4:11.PRE EOR
%   N7:17  "ms time setting to lock out inspection to give all pending images a chance to clear" %
%   T4:11  "ins 5 lock out time" %
% Rung: 5 %
SOR BST XIC B3:5/3 NXB XIC T4:11/TT BND TON T4:11 0.001 666 0 EOR
%   B3:5/3  TRACK5ERR %
%   T4:11  "ins 5 lock out time" %
% Rung: 6 %
SOR XIC B3:5/3 ONS B3:4/6 JSR U:201 EOR
%   B3:5/3  TRACK5ERR %
% Rung: 7 %
SOR XIC B3:5/3 JSR U:202 EOR
%   B3:5/3  TRACK5ERR %
% Rung: 8 %
SOR END EOR

LADDER 201 "INS5FIX1"
